// TIA Portal V20 export
// export: Created 2025-12-01T14:56:22.2948525Z, ExportSetting None, DisplayName Totally Integrated Automation Portal, DisplayVersion V20 Update 3, DisplayName TIA Portal Openness, DisplayVersion V20 Update 3, DisplayName TIA Portal Version Control Interface, DisplayVersion V20 Update 3, DisplayName STEP 7 Professional, DisplayVersion V20 Update 3, DisplayName STEP 7 Safety, DisplayVersion V20 Update 2, DisplayName WinCC Basic/Comfort/Advanced, DisplayVersion V20 Update 3, DisplayName WinCC Professional, DisplayVersion V20 Update 3, DisplayName WinCC Unified, DisplayVersion V20 Update 3
TYPE "Fuentes_Lineas"
   STRUCT
      Fuente : String[5];   // Nombre de la fuente
      Linea : Byte;   // Linea en la que esta conectada la tarjeta
      Posicion : Byte;   // posicion de la tarjeta en el cableado a partir de la fuente
   END_STRUCT;
END_TYPE
